// TIA Portal V16 export
// export: Created 2023-01-03T15:35:08.4098808Z, ExportSetting WithDefaults, DisplayName Totally Integrated Automation Portal, DisplayVersion V16, DisplayName TIA Portal Version Control Interface, DisplayVersion V16, DisplayName TIA Portal Openness, DisplayVersion V16, DisplayName STEP 7 Professional, DisplayVersion V16, DisplayName STEP 7 Safety, DisplayVersion V16, DisplayName WinCC Advanced, DisplayVersion V16
VAR_GLOBAL   // PLC tag table "Tag table_sorting station"
   "-A1" AT %M0.0 : Bool;   // return signal emergency stop ok (nc)
   "-K0" AT %M0.1 : Bool;   // main switch „ON“ (no)
   "-S0" AT %M0.2 : Bool;   // mode selector manual(0) / automatic(1)
   "-S1" AT %M0.3 : Bool;   // pushbutton automatic start (no)
   "-S2" AT %M0.4 : Bool;   // pushbutton automatic stop (nc)
   "-B1" AT %M0.5 : Bool;   // sensor cylinder -M4 retracted (no)
   "-B2" AT %M0.6 : Bool;   // sensor cylinder -M4 extended (nc)
   "-B3" AT %M0.7 : Bool;   // sensor motor -M1 actice (pulse signal for positioning) (no)
   "-B4" AT %M1.0 : Bool;   // sensor part at slide (no)
   "-B5" AT %M1.1 : Bool;   // sensor metal part (no)
   "-B6" AT %M1.2 : Bool;   // sensor part in front of cylinder -M4 (no)
   "-B7" AT %M1.3 : Bool;   // sensor part at end of conveyor (no)
   "-S3" AT %M1.4 : Bool;   // pushbutton manual mode conveyor –M1 forwards (no)
   "-S4" AT %M1.5 : Bool;   // pushbutton manual mode conveyor –M1 backwards (no)
   "-S5" AT %M1.6 : Bool;   // pushbutton manual mode cylinder -M4 retract (no)
   "-S6" AT %M1.7 : Bool;   // pushbutton manual mode cylinder -M4 extend (no)
   "-Q1" AT %M2.0 : Bool;   // conveyor motor -M1 forwards fixed speed
   "-Q2" AT %M2.1 : Bool;   // conveyor motor -M1 backwards fixed speed
   "-Q3" AT %M2.2 : Bool;   // conveyor motor -M1 variable speed
   "-M2" AT %M2.3 : Bool;   // cylinder -M4 retract
   "-M3" AT %M2.4 : Bool;   // cylinder -M4 extend
   "-P1" AT %M2.5 : Bool;   // display „main switch on“
   "-P2" AT %M2.6 : Bool;   // display „manual mode“
   "-P3" AT %M2.7 : Bool;   // display „automatic mode“
   "-P4" AT %M3.0 : Bool;   // display „emergency stop activated“
   "-P5" AT %M3.1 : Bool;   // display „automatic mode started“
   "-P6" AT %M3.2 : Bool;   // display cylinder -M4 „retracted“
   "-P7" AT %M3.3 : Bool;   // display cylinder -M4 „extended“
   "-U1" AT %MW4 : Int;   // manipulated value speed in 2 directions +/- 10V
   "-B8" AT %MW6 : Int;   // sensor actual value speed 0 …10V
   "-B9" AT %MW8 : Int;   // setpoint specification via potentiometer +/- 10V
   "-A32" AT %MW10 : Word;
   SPEED_SP AT %MD14 : Real;   // MOTOR SETPOINT IN RPM
   Ret_Val AT %M18.0 : Bool;   // Activate when speed is out of the prefered range
END_VAR
